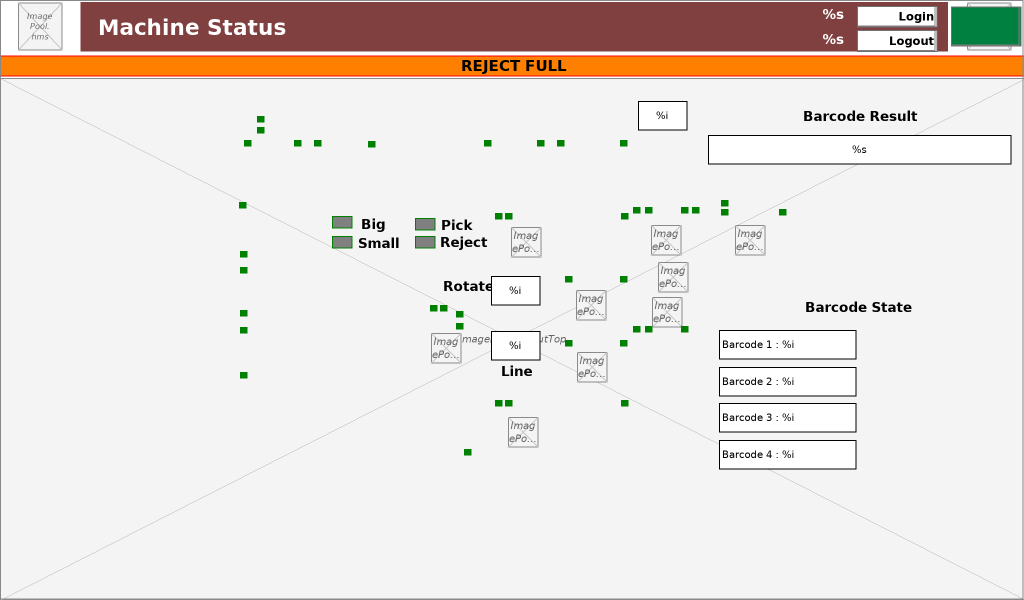
VISUALIZATION SeqStatus  // 1024x600
    Frame (0,-1 1024x55)
        shows Header()
    Label (95,15 250x25), "Machine Status"
    Image (0,78 1026x522), image: ImagePool.LayoutTop
    Image (431,333 30x30), image: ImagePool.info
        OnMouseDown: OpenDialog Dialog=PUSeq, OpenModal=True, OpenCentered=True
        OnMouseDown: execute { HMI_GVL.sCurrentJob :=  HMI_GVL.CJ_Picking; HMI_GVL.iSeqIndex   := HMI_GVL.SI_Picking; }
    Image (511,227 30x30), image: ImagePool.info
        OnMouseDown: OpenDialog Dialog=PUSeq, OpenModal=True, OpenCentered=True
        OnMouseDown: execute { HMI_GVL.sCurrentJob :=  HMI_GVL.CJ_Placing1; HMI_GVL.iSeqIndex   := HMI_GVL.SI_Placing1; }
    Image (576,290 30x30), image: ImagePool.info
        OnMouseDown: OpenDialog Dialog=PUSeq, OpenModal=True, OpenCentered=True
        OnMouseDown: execute { HMI_GVL.sCurrentJob :=  HMI_GVL.CJ_Placing2; HMI_GVL.iSeqIndex   := HMI_GVL.SI_Placing2; }
    Image (577,352 30x30), image: ImagePool.info
        OnMouseDown: OpenDialog Dialog=PUSeq, OpenModal=True, OpenCentered=True
        OnMouseDown: execute { HMI_GVL.sCurrentJob :=  HMI_GVL.CJ_Placing3; HMI_GVL.iSeqIndex   := HMI_GVL.SI_Placing3; }
    Image (508,417 30x30), image: ImagePool.info
        OnMouseDown: OpenDialog Dialog=PUSeq, OpenModal=True, OpenCentered=True
        OnMouseDown: execute { HMI_GVL.sCurrentJob :=  HMI_GVL.CJ_Placing4; HMI_GVL.iSeqIndex   := HMI_GVL.SI_Placing4; }
    Image (735,225 30x30), image: ImagePool.info
        OnMouseDown: OpenDialog Dialog=PUSeq, OpenModal=True, OpenCentered=True
        OnMouseDown: execute { HMI_GVL.sCurrentJob :=  HMI_GVL.CJ_Dispenser; HMI_GVL.iSeqIndex   := InputOutput_GVL.SeqIndexOutfeed[4]; }
    Image (652,297 30x30), image: ImagePool.info
        OnMouseDown: OpenDialog Dialog=PUSeq, OpenModal=True, OpenCentered=True
        OnMouseDown: execute { HMI_GVL.sCurrentJob :=  HMI_GVL.CJ_ShuttleEmpty; HMI_GVL.iSeqIndex   := InputOutput_GVL.SeqIndexOutfeed[1]; }
    Image (651,225 30x30), image: ImagePool.info
        OnMouseDown: OpenDialog Dialog=PUSeq, OpenModal=True, OpenCentered=True
        OnMouseDown: execute { HMI_GVL.sCurrentJob :=  HMI_GVL.CJ_ShuttleLoad; HMI_GVL.iSeqIndex   := InputOutput_GVL.SeqIndexOutfeed[2]; }
    Image (658,262 30x30), image: ImagePool.info
        OnMouseDown: OpenDialog Dialog=PUSeq, OpenModal=True, OpenCentered=True
        OnMouseDown: execute { HMI_GVL.sCurrentJob :=  HMI_GVL.CJ_ShuttleManagement; HMI_GVL.iSeqIndex   := InputOutput_GVL.SeqIndexOutfeed[3]; }
    Rectangle (415,218 20x12), colour toggle: InputOutput_GVL.xOut_Robot.Pick
    Rectangle (415,236 20x12), colour toggle: InputOutput_GVL.xOut_Robot.RejectBox
    Label (438,213 65x25), "Pick"
    Label (437,230 65x25), "Reject"
    Rectangle (456,323 7x6), colour toggle: InputOutput_GVL.xIn1405
    Rectangle (456,311 7x6), colour toggle: InputOutput_GVL.xIn1406
    Rectangle (430,305 7x6), colour toggle: InputOutput_GVL.xIn1407
    Rectangle (440,305 7x6), colour toggle: InputOutput_GVL.xIn1400
    Rectangle (633,207 7x6), colour toggle: InputOutput_GVL.Digital_Input[124]
    Rectangle (645,207 7x6), colour toggle: InputOutput_GVL.Digital_Input[122]
    Rectangle (681,207 7x6), colour toggle: InputOutput_GVL.Digital_Input[121]
    Rectangle (692,207 7x6), colour toggle: InputOutput_GVL.Digital_Input[123]
    Rectangle (633,326 7x6), colour toggle: InputOutput_GVL.Digital_Input[119]
    Rectangle (645,326 7x6), colour toggle: InputOutput_GVL.Digital_Input[117]
    Rectangle (681,326 7x6), colour toggle: InputOutput_GVL.Digital_Input[118]
    Rectangle (721,209 7x6), colour toggle: InputOutput_GVL.Digital_Input[51]
    Rectangle (721,200 7x6), colour toggle: InputOutput_GVL.Digital_Input[52]
    Rectangle (779,209 7x6), colour toggle: InputOutput_GVL.Digital_Input[50]
    Rectangle (495,400 7x6), colour toggle: InputOutput_GVL.xIn1509
    Rectangle (505,400 7x6), colour toggle: InputOutput_GVL.xIn1508
    Rectangle (621,400 7x6), colour toggle: InputOutput_GVL.xIn1507
    Rectangle (565,340 7x6), colour toggle: InputOutput_GVL.xIn1506
    Rectangle (620,340 7x6), colour toggle: InputOutput_GVL.xIn1505
    Rectangle (565,276 7x6), colour toggle: InputOutput_GVL.xIn1504
    Rectangle (620,276 7x6), colour toggle: InputOutput_GVL.xIn1503
    Rectangle (495,213 7x6), colour toggle: InputOutput_GVL.xIn1502
    Rectangle (505,213 7x6), colour toggle: InputOutput_GVL.xIn1501
    Rectangle (621,213 7x6), colour toggle: InputOutput_GVL.xIn1500
    Rectangle (620,140 7x6), colour toggle: InputOutput_GVL.Digital_Input[14]
    Rectangle (557,140 7x6), colour toggle: InputOutput_GVL.Digital_Input[15]
    Rectangle (537,140 7x6), colour toggle: InputOutput_GVL.Digital_Input[37]
    Rectangle (484,140 7x6), colour toggle: InputOutput_GVL.Digital_Input[38]
    Rectangle (368,141 7x6), colour toggle: InputOutput_GVL.Digital_Input[39]
    Rectangle (314,140 7x6), colour toggle: InputOutput_GVL.Digital_Input[40]
    Rectangle (294,140 7x6), colour toggle: InputOutput_GVL.Digital_Input[41]
    Rectangle (244,140 7x6), colour toggle: InputOutput_GVL.Digital_Input[42]
    Rectangle (239,202 7x6), colour toggle: InputOutput_GVL.Digital_Input[45]
    Rectangle (240,251 7x6), colour toggle: InputOutput_GVL.Digital_Input[46]
    Rectangle (240,267 7x6), colour toggle: InputOutput_GVL.Digital_Input[47]
    Rectangle (240,310 7x6), colour toggle: InputOutput_GVL.Digital_Input[48]
    Rectangle (240,327 7x6), colour toggle: InputOutput_GVL.Digital_Input[8]
    Rectangle (240,372 7x6), colour toggle: InputOutput_GVL.Digital_Input[9]
    Rectangle (257,127 7x6), colour toggle: InputOutput_GVL.Digital_Input[43]
    Rectangle (257,116 7x6), colour toggle: InputOutput_GVL.Digital_Input[44]
    Rectangle (464,449 7x6), colour toggle: InputOutput_GVL.xIn1005
    RoundedRectangle (638,101 49x29), "%i", text variable: InputOutput_GVL.ShuttlePosition
    Rectangle (332,216 20x12), colour toggle: InputOutput_GVL.xOut_Robot.CheckBigBox
    Label (358,212 65x25), "Big"
    Rectangle (332,236 20x12), colour toggle: InputOutput_GVL.xOut_Robot.CheckSmallBox
    Label (355,231 65x25), "Small"
    RoundedRectangle (708,135 303x29), "%s", text variable: Status_GVL.BarcodeResult
    Label (712,104 297x25), "Barcode Result"
    Label (710,295 297x25), "Barcode State"
    RoundedRectangle (719,330 137x29), "Barcode 1 : %i", text variable: InputOutput_GVL.BarcodeReader_Picking1_State
    RoundedRectangle (719,367 137x29), "Barcode 2 : %i", text variable: InputOutput_GVL.BarcodeReader_Picking2B_State
    RoundedRectangle (719,403 137x29), "Barcode 3 : %i", text variable: InputOutput_GVL.BarcodeReader_Picking3B_State
    RoundedRectangle (719,440 137x29), "Barcode 4 : %i", text variable: InputOutput_GVL.BarcodeReader_Picking4_State
    RoundedRectangle (491,331 49x29), "%i", text variable: HMI_GVL.PickLine
    Label (440,274 65x25), "Rotate"
    RoundedRectangle (491,276 49x29), "%i", text variable: InputOutput_GVL.xOut_Robot.RotatePickInt
    Label (498,359 65x25), "Line"
END_VISUALIZATION

// ---- VISUs/PLC Status/IO_Status.TcVIS
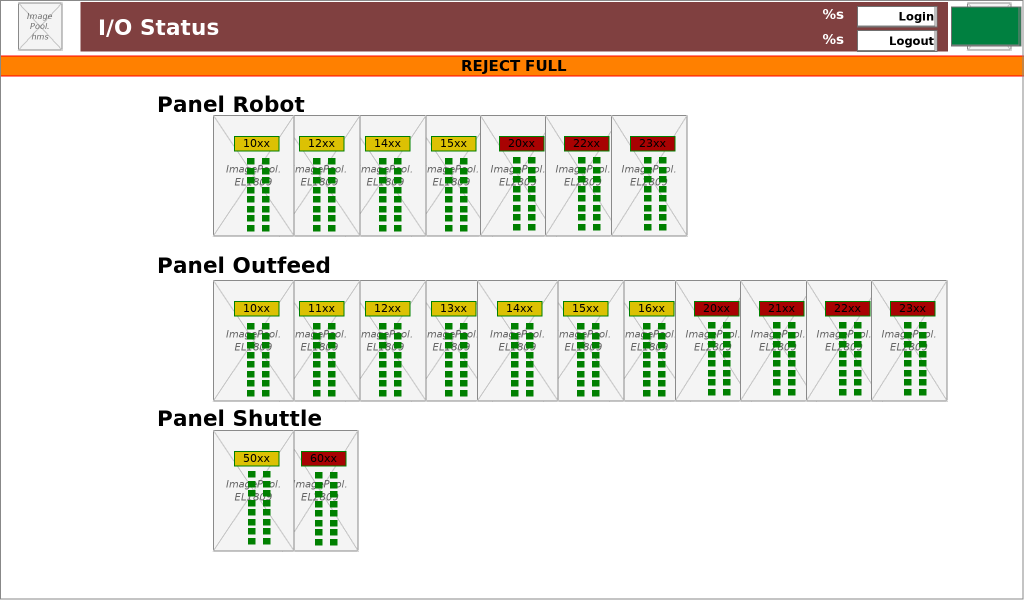
VISUALIZATION IO_Status  // 1024x600
    Image (282,430 76x121), image: ImagePool.EL2809
        OnMouseClick: OpenDialog Dialog=P3_DO1, OpenModal=True, OpenCentered=True
    Image (213,430 81x121), image: ImagePool.EL1809
        OnMouseClick: OpenDialog Dialog=P3_DI1, OpenModal=True, OpenCentered=True
    Image (411,115 81x121), image: ImagePool.EL1809
        OnMouseClick: OpenDialog Dialog=P1_DI4, OpenModal=True, OpenCentered=True
    Image (345,115 81x121), image: ImagePool.EL1809
        OnMouseClick: OpenDialog Dialog=P1_DI3, OpenModal=True, OpenCentered=True
    Image (279,115 81x121), image: ImagePool.EL1809
        OnMouseClick: OpenDialog Dialog=P1_DI2, OpenModal=True, OpenCentered=True
    Frame (0,-1 1024x55)
        shows Header()
    Label (95,15 250x25), "I/O Status"
    Image (213,115 81x121), image: ImagePool.EL1809
        OnMouseClick: OpenDialog Dialog=P1_DI1, OpenModal=True, OpenCentered=True
    Rectangle (247,158 7x6), colour toggle: InputOutput_GVL.xIn1000
    Rectangle (262,158 7x6), colour toggle: InputOutput_GVL.xIn1008
    Rectangle (247,168 7x6), colour toggle: InputOutput_GVL.xIn1001
    Rectangle (262,168 7x6), colour toggle: InputOutput_GVL.xIn1009
    Rectangle (247,177 7x6), colour toggle: InputOutput_GVL.xIn1002
    Rectangle (262,177 7x6), colour toggle: InputOutput_GVL.xIn1010
    Rectangle (247,187 7x6), colour toggle: InputOutput_GVL.xIn1003
    Rectangle (262,187 7x6), colour toggle: InputOutput_GVL.xIn1011
    Rectangle (247,196 7x6), colour toggle: InputOutput_GVL.xIn1004
    Rectangle (262,196 7x6), colour toggle: InputOutput_GVL.xIn1012
    Rectangle (247,206 7x6), colour toggle: InputOutput_GVL.xIn1005
    Rectangle (262,206 7x6), colour toggle: InputOutput_GVL.xIn1013
    Rectangle (247,215 7x6), colour toggle: InputOutput_GVL.xIn1006
    Rectangle (262,215 7x6), colour toggle: InputOutput_GVL.xIn1014
    Rectangle (247,225 7x6), colour toggle: InputOutput_GVL.xIn1007
    Rectangle (262,225 7x6), colour toggle: InputOutput_GVL.xIn1015
    Label (237,134 37x20), "10xx"
    Rectangle (313,158 7x6), colour toggle: InputOutput_GVL.xIn1200
    Rectangle (328,158 7x6), colour toggle: InputOutput_GVL.xIn1208
    Rectangle (313,168 7x6), colour toggle: InputOutput_GVL.xIn1201
    Rectangle (328,168 7x6), colour toggle: InputOutput_GVL.xIn1209
    Rectangle (313,177 7x6), colour toggle: InputOutput_GVL.xIn1202
    Rectangle (328,177 7x6), colour toggle: InputOutput_GVL.xIn1210
    Rectangle (313,187 7x6), colour toggle: InputOutput_GVL.xIn1203
    Rectangle (328,187 7x6), colour toggle: InputOutput_GVL.xIn1211
    Rectangle (313,196 7x6), colour toggle: InputOutput_GVL.xIn1204
    Rectangle (328,196 7x6), colour toggle: InputOutput_GVL.xIn1212
    Rectangle (313,206 7x6), colour toggle: InputOutput_GVL.xIn1205
    Rectangle (328,206 7x6), colour toggle: InputOutput_GVL.xIn1213
    Rectangle (313,215 7x6), colour toggle: InputOutput_GVL.xIn1206
    Rectangle (328,215 7x6), colour toggle: InputOutput_GVL.xIn1214
    Rectangle (313,225 7x6), colour toggle: InputOutput_GVL.xIn1207
    Rectangle (328,225 7x6), colour toggle: InputOutput_GVL.xIn1215
    Rectangle (379,158 7x6), colour toggle: InputOutput_GVL.xIn1400
    Rectangle (394,158 7x6), colour toggle: InputOutput_GVL.xIn1408
    Rectangle (379,168 7x6), colour toggle: InputOutput_GVL.xIn1401
    Rectangle (394,168 7x6), colour toggle: InputOutput_GVL.xIn1409
    Rectangle (379,177 7x6), colour toggle: InputOutput_GVL.xIn1402
    Rectangle (394,177 7x6), colour toggle: InputOutput_GVL.xIn1410
    Rectangle (379,187 7x6), colour toggle: InputOutput_GVL.xIn1403
    Rectangle (394,187 7x6), colour toggle: InputOutput_GVL.xIn1411
    Rectangle (379,196 7x6), colour toggle: InputOutput_GVL.xIn1404
    Rectangle (394,196 7x6), colour toggle: InputOutput_GVL.xIn1412
    Rectangle (379,206 7x6), colour toggle: InputOutput_GVL.xIn1405
    Rectangle (394,206 7x6), colour toggle: InputOutput_GVL.xIn1413
    Rectangle (379,215 7x6), colour toggle: InputOutput_GVL.xIn1406
    Rectangle (394,215 7x6), colour toggle: InputOutput_GVL.xIn1414
    Rectangle (379,225 7x6), colour toggle: InputOutput_GVL.xIn1407
    Rectangle (394,225 7x6), colour toggle: InputOutput_GVL.xIn1415
    Rectangle (445,158 7x6), colour toggle: InputOutput_GVL.xIn1500
    Rectangle (460,158 7x6), colour toggle: InputOutput_GVL.xIn1508
    Rectangle (445,168 7x6), colour toggle: InputOutput_GVL.xIn1501
    Rectangle (460,168 7x6), colour toggle: InputOutput_GVL.xIn1509
    Rectangle (445,177 7x6), colour toggle: InputOutput_GVL.xIn1502
    Rectangle (460,177 7x6), colour toggle: InputOutput_GVL.xIn1510
    Rectangle (445,187 7x6), colour toggle: InputOutput_GVL.xIn1503
    Rectangle (460,187 7x6), colour toggle: InputOutput_GVL.xIn1511
    Rectangle (445,196 7x6), colour toggle: InputOutput_GVL.xIn1504
    Rectangle (460,196 7x6), colour toggle: InputOutput_GVL.xIn1512
    Rectangle (445,206 7x6), colour toggle: InputOutput_GVL.xIn1505
    Rectangle (460,206 7x6), colour toggle: InputOutput_GVL.xIn1513
    Rectangle (445,215 7x6), colour toggle: InputOutput_GVL.xIn1506
    Rectangle (460,215 7x6), colour toggle: InputOutput_GVL.xIn1514
    Rectangle (445,225 7x6), colour toggle: InputOutput_GVL.xIn1507
    Rectangle (460,225 7x6), colour toggle: InputOutput_GVL.xIn1515
    Rectangle (234,136 45x15), "10xx", colour toggle: HMI_GVL.xOut_HMI_Status_EcSlave[1]
    Rectangle (299,136 45x15), "12xx", colour toggle: HMI_GVL.xOut_HMI_Status_EcSlave[2]
    Rectangle (365,136 45x15), "14xx", colour toggle: HMI_GVL.xOut_HMI_Status_EcSlave[3]
    Rectangle (431,136 45x15), "15xx", colour toggle: HMI_GVL.xOut_HMI_Status_EcSlave[4]
    Image (480,115 76x121), image: ImagePool.EL2809
        OnMouseClick: OpenDialog Dialog=P1_DO1, OpenModal=True, OpenCentered=True
    Rectangle (513,157 7x6), colour toggle: InputOutput_GVL.xOut2000
    Rectangle (528,157 7x6), colour toggle: InputOutput_GVL.xOut2008
    Rectangle (513,167 7x6), colour toggle: InputOutput_GVL.xOut2001
    Rectangle (528,167 7x6), colour toggle: InputOutput_GVL.xOut2009
    Rectangle (513,176 7x6), colour toggle: InputOutput_GVL.xOut2002
    Rectangle (528,176 7x6), colour toggle: InputOutput_GVL.xOut2010
    Rectangle (513,186 7x6), colour toggle: InputOutput_GVL.xOut2003
    Rectangle (528,186 7x6), colour toggle: InputOutput_GVL.xOut2011
    Rectangle (513,195 7x6), colour toggle: InputOutput_GVL.xOut2004
    Rectangle (528,195 7x6), colour toggle: InputOutput_GVL.xOut2012
    Rectangle (513,205 7x6), colour toggle: InputOutput_GVL.xOut2005
    Rectangle (528,205 7x6), colour toggle: InputOutput_GVL.xOut2013
    Rectangle (513,214 7x6), colour toggle: InputOutput_GVL.xOut2006
    Rectangle (528,214 7x6), colour toggle: InputOutput_GVL.xOut2014
    Rectangle (513,224 7x6), colour toggle: InputOutput_GVL.xOut2007
    Rectangle (528,224 7x6), colour toggle: InputOutput_GVL.xOut2015
    Label (502,136 37x20), "10xx"
    Rectangle (499,136 45x15), "20xx", colour toggle: HMI_GVL.xOut_HMI_Status_EcSlave[5]
    Image (545,115 76x121), image: ImagePool.EL2809
        OnMouseClick: OpenDialog Dialog=P1_DO2, OpenModal=True, OpenCentered=True
    Rectangle (578,157 7x6), colour toggle: InputOutput_GVL.xOut2200
    Rectangle (593,157 7x6), colour toggle: InputOutput_GVL.xOut2208
    Rectangle (578,167 7x6), colour toggle: InputOutput_GVL.xOut2201
    Rectangle (593,167 7x6), colour toggle: InputOutput_GVL.xOut2209
    Rectangle (578,176 7x6), colour toggle: InputOutput_GVL.xOut2202
    Rectangle (593,176 7x6), colour toggle: InputOutput_GVL.xOut2210
    Rectangle (578,186 7x6), colour toggle: InputOutput_GVL.xOut2203
    Rectangle (593,186 7x6), colour toggle: InputOutput_GVL.xOut2211
    Rectangle (578,195 7x6), colour toggle: InputOutput_GVL.xOut2204
    Rectangle (593,195 7x6), colour toggle: InputOutput_GVL.xOut2212
    Rectangle (578,205 7x6), colour toggle: InputOutput_GVL.xOut2205
    Rectangle (593,205 7x6), colour toggle: InputOutput_GVL.xOut2213
    Rectangle (578,214 7x6), colour toggle: InputOutput_GVL.xOut2206
    Rectangle (593,214 7x6), colour toggle: InputOutput_GVL.xOut2214
    Rectangle (578,224 7x6), colour toggle: InputOutput_GVL.xOut2207
    Rectangle (593,224 7x6), colour toggle: InputOutput_GVL.xOut2215
    Label (567,135 37x20), "10xx"
    Rectangle (564,136 45x15), "22xx", colour toggle: HMI_GVL.xOut_HMI_Status_EcSlave[6]
    Image (611,115 76x121), image: ImagePool.EL2809
        OnMouseClick: OpenDialog Dialog=P1_DO3, OpenModal=True, OpenCentered=True
    Rectangle (644,157 7x6), colour toggle: InputOutput_GVL.xOut2300
    Rectangle (659,157 7x6), colour toggle: InputOutput_GVL.xOut2308
    Rectangle (644,167 7x6), colour toggle: InputOutput_GVL.xOut2301
    Rectangle (659,167 7x6), colour toggle: InputOutput_GVL.xOut2309
    Rectangle (644,176 7x6), colour toggle: InputOutput_GVL.xOut2302
    Rectangle (659,176 7x6), colour toggle: InputOutput_GVL.xOut2310
    Rectangle (644,186 7x6), colour toggle: InputOutput_GVL.xOut2303
    Rectangle (659,186 7x6), colour toggle: InputOutput_GVL.xOut2311
    Rectangle (644,195 7x6), colour toggle: InputOutput_GVL.xOut2304
    Rectangle (659,195 7x6), colour toggle: InputOutput_GVL.xOut2312
    Rectangle (644,205 7x6), colour toggle: InputOutput_GVL.xOut2305
    Rectangle (659,205 7x6), colour toggle: InputOutput_GVL.xOut2313
    Rectangle (644,214 7x6), colour toggle: InputOutput_GVL.xOut2306
    Rectangle (659,214 7x6), colour toggle: InputOutput_GVL.xOut2314
    Rectangle (644,224 7x6), colour toggle: InputOutput_GVL.xOut2307
    Rectangle (659,224 7x6), colour toggle: InputOutput_GVL.xOut2315
    Label (633,135 37x20), "10xx"
    Rectangle (630,136 45x15), "23xx", colour toggle: HMI_GVL.xOut_HMI_Status_EcSlave[7]
    Label (154,92 250x25), "Panel Robot"
    Label (154,253 250x25), "Panel Outfeed"
    Rectangle (248,471 7x6), colour toggle: InputOutput_GVL.Digital_Input[113]
    Rectangle (263,471 7x6), colour toggle: InputOutput_GVL.Digital_Input[121]
    Rectangle (248,481 7x6), colour toggle: InputOutput_GVL.Digital_Input[114]
    Rectangle (263,481 7x6), colour toggle: InputOutput_GVL.Digital_Input[122]
    Rectangle (248,490 7x6), colour toggle: InputOutput_GVL.Digital_Input[115]
    Rectangle (263,490 7x6), colour toggle: InputOutput_GVL.Digital_Input[123]
    Rectangle (248,500 7x6), colour toggle: InputOutput_GVL.Digital_Input[116]
    Rectangle (263,500 7x6), colour toggle: InputOutput_GVL.Digital_Input[124]
    Rectangle (248,509 7x6), colour toggle: InputOutput_GVL.Digital_Input[117]
    Rectangle (263,509 7x6), colour toggle: InputOutput_GVL.Digital_Input[125]
    Rectangle (248,519 7x6), colour toggle: InputOutput_GVL.Digital_Input[118]
    Rectangle (263,519 7x6), colour toggle: InputOutput_GVL.Digital_Input[126]
    Rectangle (248,528 7x6), colour toggle: InputOutput_GVL.Digital_Input[119]
    Rectangle (263,528 7x6), colour toggle: InputOutput_GVL.Digital_Input[127]
    Rectangle (248,538 7x6), colour toggle: InputOutput_GVL.Digital_Input[120]
    Rectangle (263,538 7x6), colour toggle: InputOutput_GVL.Digital_Input[128]
    Label (237,448 37x20), "10xx"
    Rectangle (234,451 45x15), "50xx", colour toggle: HMI_GVL.xOut_HMI_Status_EcSlave[1]
    Rectangle (315,472 7x6), colour toggle: InputOutput_GVL.Digital_Output[65]
    Rectangle (330,472 7x6), colour toggle: InputOutput_GVL.Digital_Output[73]
    Rectangle (315,482 7x6), colour toggle: InputOutput_GVL.Digital_Output[66]
    Rectangle (330,482 7x6), colour toggle: InputOutput_GVL.Digital_Output[74]
    Rectangle (315,491 7x6), colour toggle: InputOutput_GVL.Digital_Output[67]
    Rectangle (330,491 7x6), colour toggle: InputOutput_GVL.Digital_Output[75]
    Rectangle (315,501 7x6), colour toggle: InputOutput_GVL.Digital_Output[68]
    Rectangle (330,501 7x6), colour toggle: InputOutput_GVL.Digital_Output[76]
    Rectangle (315,510 7x6), colour toggle: InputOutput_GVL.Digital_Output[69]
    Rectangle (330,510 7x6), colour toggle: InputOutput_GVL.Digital_Output[77]
    Rectangle (315,520 7x6), colour toggle: InputOutput_GVL.Digital_Output[70]
    Rectangle (330,520 7x6), colour toggle: InputOutput_GVL.Digital_Output[78]
    Rectangle (315,529 7x6), colour toggle: InputOutput_GVL.Digital_Output[71]
    Rectangle (330,529 7x6), colour toggle: InputOutput_GVL.Digital_Output[79]
    Rectangle (315,539 7x6), colour toggle: InputOutput_GVL.Digital_Output[72]
    Rectangle (330,539 7x6), colour toggle: InputOutput_GVL.Digital_Output[80]
    Label (304,450 37x20), "10xx"
    Rectangle (301,451 45x15), "60xx", colour toggle: HMI_GVL.xOut_HMI_Status_EcSlave[1]
    Label (154,406 250x25), "Panel Shuttle"
    Image (411,280 81x121), image: ImagePool.EL1809
        OnMouseClick: OpenDialog Dialog=P2_DI4, OpenModal=True, OpenCentered=True
    Image (345,280 81x121), image: ImagePool.EL1809
        OnMouseClick: OpenDialog Dialog=P2_DI3, OpenModal=True, OpenCentered=True
    Image (279,280 81x121), image: ImagePool.EL1809
        OnMouseClick: OpenDialog Dialog=P2_DI2, OpenModal=True, OpenCentered=True
    Image (213,280 81x121), image: ImagePool.EL1809
        OnMouseClick: OpenDialog Dialog=P2_DI1, OpenModal=True, OpenCentered=True
    Rectangle (247,323 7x6), colour toggle: InputOutput_GVL.Digital_Input[1]
    Rectangle (262,323 7x6), colour toggle: InputOutput_GVL.Digital_Input[9]
    Rectangle (247,333 7x6), colour toggle: InputOutput_GVL.Digital_Input[2]
    Rectangle (262,333 7x6), colour toggle: InputOutput_GVL.Digital_Input[10]
    Rectangle (247,342 7x6), colour toggle: InputOutput_GVL.Digital_Input[3]
    Rectangle (262,342 7x6), colour toggle: InputOutput_GVL.Digital_Input[11]
    Rectangle (247,352 7x6), colour toggle: InputOutput_GVL.Digital_Input[4]
    Rectangle (262,352 7x6), colour toggle: InputOutput_GVL.Digital_Input[12]
    Rectangle (247,361 7x6), colour toggle: InputOutput_GVL.Digital_Input[5]
    Rectangle (262,361 7x6), colour toggle: InputOutput_GVL.Digital_Input[13]
    Rectangle (247,371 7x6), colour toggle: InputOutput_GVL.Digital_Input[6]
    Rectangle (262,371 7x6), colour toggle: InputOutput_GVL.Digital_Input[14]
    Rectangle (247,380 7x6), colour toggle: InputOutput_GVL.Digital_Input[7]
    Rectangle (262,380 7x6), colour toggle: InputOutput_GVL.Digital_Input[15]
    Rectangle (247,390 7x6), colour toggle: InputOutput_GVL.Digital_Input[8]
    Rectangle (262,390 7x6), colour toggle: InputOutput_GVL.Digital_Input[16]
    Label (237,299 37x20), "10xx"
    Rectangle (313,323 7x6), colour toggle: InputOutput_GVL.Digital_Input[17]
    Rectangle (328,323 7x6), colour toggle: InputOutput_GVL.Digital_Input[25]
    Rectangle (313,333 7x6), colour toggle: InputOutput_GVL.Digital_Input[18]
    Rectangle (328,333 7x6), colour toggle: InputOutput_GVL.Digital_Input[26]
    Rectangle (313,342 7x6), colour toggle: InputOutput_GVL.Digital_Input[19]
    Rectangle (328,342 7x6), colour toggle: InputOutput_GVL.Digital_Input[27]
    Rectangle (313,352 7x6), colour toggle: InputOutput_GVL.Digital_Input[20]
    Rectangle (328,352 7x6), colour toggle: InputOutput_GVL.Digital_Input[28]
    Rectangle (313,361 7x6), colour toggle: InputOutput_GVL.Digital_Input[21]
    Rectangle (328,361 7x6), colour toggle: InputOutput_GVL.Digital_Input[29]
    Rectangle (313,371 7x6), colour toggle: InputOutput_GVL.Digital_Input[22]
    Rectangle (328,371 7x6), colour toggle: InputOutput_GVL.Digital_Input[30]
    Rectangle (313,380 7x6), colour toggle: InputOutput_GVL.Digital_Input[23]
    Rectangle (328,380 7x6), colour toggle: InputOutput_GVL.Digital_Input[31]
    Rectangle (313,390 7x6), colour toggle: InputOutput_GVL.Digital_Input[24]
    Rectangle (328,390 7x6), colour toggle: InputOutput_GVL.Digital_Input[32]
    Rectangle (379,323 7x6), colour toggle: InputOutput_GVL.Digital_Input[33]
    Rectangle (394,323 7x6), colour toggle: InputOutput_GVL.Digital_Input[41]
    Rectangle (379,333 7x6), colour toggle: InputOutput_GVL.Digital_Input[34]
    Rectangle (394,333 7x6), colour toggle: InputOutput_GVL.Digital_Input[42]
    Rectangle (379,342 7x6), colour toggle: InputOutput_GVL.Digital_Input[35]
    Rectangle (394,342 7x6), colour toggle: InputOutput_GVL.Digital_Input[43]
    Rectangle (379,352 7x6), colour toggle: InputOutput_GVL.Digital_Input[36]
    Rectangle (394,352 7x6), colour toggle: InputOutput_GVL.Digital_Input[44]
    Rectangle (379,361 7x6), colour toggle: InputOutput_GVL.Digital_Input[37]
    Rectangle (394,361 7x6), colour toggle: InputOutput_GVL.Digital_Input[45]
    Rectangle (379,371 7x6), colour toggle: InputOutput_GVL.Digital_Input[38]
    Rectangle (394,371 7x6), colour toggle: InputOutput_GVL.Digital_Input[46]
    Rectangle (379,380 7x6), colour toggle: InputOutput_GVL.Digital_Input[39]
    Rectangle (394,380 7x6), colour toggle: InputOutput_GVL.Digital_Input[47]
    Rectangle (379,390 7x6), colour toggle: InputOutput_GVL.Digital_Input[40]
    Rectangle (394,390 7x6), colour toggle: InputOutput_GVL.Digital_Input[48]
    Rectangle (445,323 7x6), colour toggle: InputOutput_GVL.Digital_Input[49]
    Rectangle (460,323 7x6), colour toggle: InputOutput_GVL.Digital_Input[57]
    Rectangle (445,333 7x6), colour toggle: InputOutput_GVL.Digital_Input[50]
    Rectangle (460,333 7x6), colour toggle: InputOutput_GVL.Digital_Input[58]
    Rectangle (445,342 7x6), colour toggle: InputOutput_GVL.Digital_Input[51]
    Rectangle (460,342 7x6), colour toggle: InputOutput_GVL.Digital_Input[59]
    Rectangle (445,352 7x6), colour toggle: InputOutput_GVL.Digital_Input[52]
    Rectangle (460,352 7x6), colour toggle: InputOutput_GVL.Digital_Input[60]
    Rectangle (445,361 7x6), colour toggle: InputOutput_GVL.Digital_Input[53]
    Rectangle (460,361 7x6), colour toggle: InputOutput_GVL.Digital_Input[61]
    Rectangle (445,371 7x6), colour toggle: InputOutput_GVL.Digital_Input[54]
    Rectangle (460,371 7x6), colour toggle: InputOutput_GVL.Digital_Input[62]
    Rectangle (445,380 7x6), colour toggle: InputOutput_GVL.Digital_Input[55]
    Rectangle (460,380 7x6), colour toggle: InputOutput_GVL.Digital_Input[63]
    Rectangle (445,390 7x6), colour toggle: InputOutput_GVL.Digital_Input[56]
    Rectangle (460,390 7x6), colour toggle: InputOutput_GVL.Digital_Input[64]
    Rectangle (234,301 45x15), "10xx", colour toggle: HMI_GVL.xOut_HMI_Status_EcSlave[1]
    Rectangle (299,301 45x15), "11xx", colour toggle: HMI_GVL.xOut_HMI_Status_EcSlave[2]
    Rectangle (365,301 45x15), "12xx", colour toggle: HMI_GVL.xOut_HMI_Status_EcSlave[3]
    Rectangle (431,301 45x15), "13xx", colour toggle: HMI_GVL.xOut_HMI_Status_EcSlave[4]
    Image (609,280 81x121), image: ImagePool.EL1809
        OnMouseClick: OpenDialog Dialog=P2_DI7, OpenModal=True, OpenCentered=True
    Image (543,280 81x121), image: ImagePool.EL1809
        OnMouseClick: OpenDialog Dialog=P2_DI6, OpenModal=True, OpenCentered=True
    Image (477,280 81x121), image: ImagePool.EL1809
        OnMouseClick: OpenDialog Dialog=P2_DI5, OpenModal=True, OpenCentered=True
    Rectangle (511,323 7x6), colour toggle: InputOutput_GVL.Digital_Input[65]
    Rectangle (526,323 7x6), colour toggle: InputOutput_GVL.Digital_Input[73]
    Rectangle (511,333 7x6), colour toggle: InputOutput_GVL.Digital_Input[66]
    Rectangle (526,333 7x6), colour toggle: InputOutput_GVL.Digital_Input[74]
    Rectangle (511,342 7x6), colour toggle: InputOutput_GVL.Digital_Input[67]
    Rectangle (526,342 7x6), colour toggle: InputOutput_GVL.Digital_Input[75]
    Rectangle (511,352 7x6), colour toggle: InputOutput_GVL.Digital_Input[68]
    Rectangle (526,352 7x6), colour toggle: InputOutput_GVL.Digital_Input[76]
    Rectangle (511,361 7x6), colour toggle: InputOutput_GVL.Digital_Input[69]
    Rectangle (526,361 7x6), colour toggle: InputOutput_GVL.Digital_Input[77]
    Rectangle (511,371 7x6), colour toggle: InputOutput_GVL.Digital_Input[70]
    Rectangle (526,371 7x6), colour toggle: InputOutput_GVL.Digital_Input[78]
    Rectangle (511,380 7x6), colour toggle: InputOutput_GVL.Digital_Input[71]
    Rectangle (526,380 7x6), colour toggle: InputOutput_GVL.Digital_Input[79]
    Rectangle (511,390 7x6), colour toggle: InputOutput_GVL.Digital_Input[72]
    Rectangle (526,390 7x6), colour toggle: InputOutput_GVL.Digital_Input[80]
    Rectangle (577,323 7x6), colour toggle: InputOutput_GVL.Digital_Input[81]
    Rectangle (592,323 7x6), colour toggle: InputOutput_GVL.Digital_Input[89]
    Rectangle (577,333 7x6), colour toggle: InputOutput_GVL.Digital_Input[82]
    Rectangle (592,333 7x6), colour toggle: InputOutput_GVL.Digital_Input[90]
    Rectangle (577,342 7x6), colour toggle: InputOutput_GVL.Digital_Input[83]
    Rectangle (592,342 7x6), colour toggle: InputOutput_GVL.Digital_Input[91]
    Rectangle (577,352 7x6), colour toggle: InputOutput_GVL.Digital_Input[84]
    Rectangle (592,352 7x6), colour toggle: InputOutput_GVL.Digital_Input[92]
    Rectangle (577,361 7x6), colour toggle: InputOutput_GVL.Digital_Input[85]
    Rectangle (592,361 7x6), colour toggle: InputOutput_GVL.Digital_Input[93]
    Rectangle (577,371 7x6), colour toggle: InputOutput_GVL.Digital_Input[86]
    Rectangle (592,371 7x6), colour toggle: InputOutput_GVL.Digital_Input[94]
    Rectangle (577,380 7x6), colour toggle: InputOutput_GVL.Digital_Input[87]
    Rectangle (592,380 7x6), colour toggle: InputOutput_GVL.Digital_Input[95]
    Rectangle (577,390 7x6), colour toggle: InputOutput_GVL.Digital_Input[88]
    Rectangle (592,390 7x6), colour toggle: InputOutput_GVL.Digital_Input[96]
    Rectangle (643,323 7x6), colour toggle: InputOutput_GVL.Digital_Input[97]
    Rectangle (658,323 7x6), colour toggle: InputOutput_GVL.Digital_Input[105]
    Rectangle (643,333 7x6), colour toggle: InputOutput_GVL.Digital_Input[98]
    Rectangle (658,333 7x6), colour toggle: InputOutput_GVL.Digital_Input[106]
    Rectangle (643,342 7x6), colour toggle: InputOutput_GVL.Digital_Input[99]
    Rectangle (658,342 7x6), colour toggle: InputOutput_GVL.Digital_Input[107]
    Rectangle (643,352 7x6), colour toggle: InputOutput_GVL.Digital_Input[100]
    Rectangle (658,352 7x6), colour toggle: InputOutput_GVL.Digital_Input[108]
    Rectangle (643,361 7x6), colour toggle: InputOutput_GVL.Digital_Input[101]
    Rectangle (658,361 7x6), colour toggle: InputOutput_GVL.Digital_Input[109]
    Rectangle (643,371 7x6), colour toggle: InputOutput_GVL.Digital_Input[102]
    Rectangle (658,371 7x6), colour toggle: InputOutput_GVL.Digital_Input[110]
    Rectangle (643,380 7x6), colour toggle: InputOutput_GVL.Digital_Input[103]
    Rectangle (658,380 7x6), colour toggle: InputOutput_GVL.Digital_Input[111]
    Rectangle (643,390 7x6), colour toggle: InputOutput_GVL.Digital_Input[104]
    Rectangle (658,390 7x6), colour toggle: InputOutput_GVL.Digital_Input[112]
    Rectangle (497,301 45x15), "14xx", colour toggle: HMI_GVL.xOut_HMI_Status_EcSlave[2]
    Rectangle (563,301 45x15), "15xx", colour toggle: HMI_GVL.xOut_HMI_Status_EcSlave[3]
    Rectangle (629,301 45x15), "16xx", colour toggle: HMI_GVL.xOut_HMI_Status_EcSlave[4]
    Image (675,280 76x121), image: ImagePool.EL2809
        OnMouseClick: OpenDialog Dialog=P2_DO1, OpenModal=True, OpenCentered=True
    Rectangle (708,322 7x6), colour toggle: InputOutput_GVL.Digital_Output[1]
    Rectangle (723,322 7x6), colour toggle: InputOutput_GVL.Digital_Output[9]
    Rectangle (708,332 7x6), colour toggle: InputOutput_GVL.Digital_Output[2]
    Rectangle (723,332 7x6), colour toggle: InputOutput_GVL.Digital_Output[10]
    Rectangle (708,341 7x6), colour toggle: InputOutput_GVL.Digital_Output[3]
    Rectangle (723,341 7x6), colour toggle: InputOutput_GVL.Digital_Output[11]
    Rectangle (708,351 7x6), colour toggle: InputOutput_GVL.Digital_Output[4]
    Rectangle (723,351 7x6), colour toggle: InputOutput_GVL.Digital_Output[12]
    Rectangle (708,360 7x6), colour toggle: InputOutput_GVL.Digital_Output[5]
    Rectangle (723,360 7x6), colour toggle: InputOutput_GVL.Digital_Output[13]
    Rectangle (708,370 7x6), colour toggle: InputOutput_GVL.Digital_Output[6]
    Rectangle (723,370 7x6), colour toggle: InputOutput_GVL.Digital_Output[14]
    Rectangle (708,379 7x6), colour toggle: InputOutput_GVL.Digital_Output[7]
    Rectangle (723,379 7x6), colour toggle: InputOutput_GVL.Digital_Output[15]
    Rectangle (708,389 7x6), colour toggle: InputOutput_GVL.Digital_Output[8]
    Rectangle (723,389 7x6), colour toggle: InputOutput_GVL.Digital_Output[16]
    Label (697,301 37x20), "10xx"
    Rectangle (694,301 45x15), "20xx", colour toggle: HMI_GVL.xOut_HMI_Status_EcSlave[1]
    Image (740,280 76x121), image: ImagePool.EL2809
        OnMouseClick: OpenDialog Dialog=P2_DO2, OpenModal=True, OpenCentered=True
    Rectangle (773,322 7x6), colour toggle: InputOutput_GVL.Digital_Output[17]
    Rectangle (788,322 7x6), colour toggle: InputOutput_GVL.Digital_Output[25]
    Rectangle (773,332 7x6), colour toggle: InputOutput_GVL.Digital_Output[18]
    Rectangle (788,332 7x6), colour toggle: InputOutput_GVL.Digital_Output[26]
    Rectangle (773,341 7x6), colour toggle: InputOutput_GVL.Digital_Output[19]
    Rectangle (788,341 7x6), colour toggle: InputOutput_GVL.Digital_Output[27]
    Rectangle (773,351 7x6), colour toggle: InputOutput_GVL.Digital_Output[20]
    Rectangle (788,351 7x6), colour toggle: InputOutput_GVL.Digital_Output[28]
    Rectangle (773,360 7x6), colour toggle: InputOutput_GVL.Digital_Output[21]
    Rectangle (788,360 7x6), colour toggle: InputOutput_GVL.Digital_Output[29]
    Rectangle (773,370 7x6), colour toggle: InputOutput_GVL.Digital_Output[22]
    Rectangle (788,370 7x6), colour toggle: InputOutput_GVL.Digital_Output[30]
    Rectangle (773,379 7x6), colour toggle: InputOutput_GVL.Digital_Output[23]
    Rectangle (788,379 7x6), colour toggle: InputOutput_GVL.Digital_Output[31]
    Rectangle (773,389 7x6), colour toggle: InputOutput_GVL.Digital_Output[24]
    Rectangle (788,389 7x6), colour toggle: InputOutput_GVL.Digital_Output[32]
    Label (762,300 37x20), "10xx"
    Rectangle (759,301 45x15), "21xx", colour toggle: HMI_GVL.xOut_HMI_Status_EcSlave[1]
    Image (806,280 76x121), image: ImagePool.EL2809
        OnMouseClick: OpenDialog Dialog=P2_DO3, OpenModal=True, OpenCentered=True
    Rectangle (839,322 7x6), colour toggle: InputOutput_GVL.Digital_Output[33]
    Rectangle (854,322 7x6), colour toggle: InputOutput_GVL.Digital_Output[41]
    Rectangle (839,332 7x6), colour toggle: InputOutput_GVL.Digital_Output[34]
    Rectangle (854,332 7x6), colour toggle: InputOutput_GVL.Digital_Output[42]
    Rectangle (839,341 7x6), colour toggle: InputOutput_GVL.Digital_Output[35]
    Rectangle (854,341 7x6), colour toggle: InputOutput_GVL.Digital_Output[43]
    Rectangle (839,351 7x6), colour toggle: InputOutput_GVL.Digital_Output[36]
    Rectangle (854,351 7x6), colour toggle: InputOutput_GVL.Digital_Output[44]
    Rectangle (839,360 7x6), colour toggle: InputOutput_GVL.Digital_Output[37]
    Rectangle (854,360 7x6), colour toggle: InputOutput_GVL.Digital_Output[45]
    Rectangle (839,370 7x6), colour toggle: InputOutput_GVL.Digital_Output[38]
    Rectangle (854,370 7x6), colour toggle: InputOutput_GVL.Digital_Output[46]
    Rectangle (839,379 7x6), colour toggle: InputOutput_GVL.Digital_Output[39]
    Rectangle (854,379 7x6), colour toggle: InputOutput_GVL.Digital_Output[47]
    Rectangle (839,389 7x6), colour toggle: InputOutput_GVL.Digital_Output[40]
    Rectangle (854,389 7x6), colour toggle: InputOutput_GVL.Digital_Output[48]
    Label (828,300 37x20), "10xx"
    Rectangle (825,301 45x15), "22xx", colour toggle: HMI_GVL.xOut_HMI_Status_EcSlave[1]
    Image (871,280 76x121), image: ImagePool.EL2809
        OnMouseClick: OpenDialog Dialog=P2_DO4, OpenModal=True, OpenCentered=True
    Rectangle (904,322 7x6), colour toggle: InputOutput_GVL.Digital_Output[49]
    Rectangle (919,322 7x6), colour toggle: InputOutput_GVL.Digital_Output[57]
    Rectangle (904,332 7x6), colour toggle: InputOutput_GVL.Digital_Output[50]
    Rectangle (919,332 7x6), colour toggle: InputOutput_GVL.Digital_Output[58]
    Rectangle (904,341 7x6), colour toggle: InputOutput_GVL.Digital_Output[51]
    Rectangle (919,341 7x6), colour toggle: InputOutput_GVL.Digital_Output[59]
    Rectangle (904,351 7x6), colour toggle: InputOutput_GVL.Digital_Output[52]
    Rectangle (919,351 7x6), colour toggle: InputOutput_GVL.Digital_Output[60]
    Rectangle (904,360 7x6), colour toggle: InputOutput_GVL.Digital_Output[53]
    Rectangle (919,360 7x6), colour toggle: InputOutput_GVL.Digital_Output[61]
    Rectangle (904,370 7x6), colour toggle: InputOutput_GVL.Digital_Output[54]
    Rectangle (919,370 7x6), colour toggle: InputOutput_GVL.Digital_Output[62]
    Rectangle (904,379 7x6), colour toggle: InputOutput_GVL.Digital_Output[55]
    Rectangle (919,379 7x6), colour toggle: InputOutput_GVL.Digital_Output[63]
    Rectangle (904,389 7x6), colour toggle: InputOutput_GVL.Digital_Output[56]
    Rectangle (919,389 7x6), colour toggle: InputOutput_GVL.Digital_Output[64]
    Label (893,300 37x20), "10xx"
    Rectangle (890,301 45x15), "23xx", colour toggle: HMI_GVL.xOut_HMI_Status_EcSlave[1]
END_VISUALIZATION

// ---- VISUs/TestMode/Test_Outfeed.TcVIS
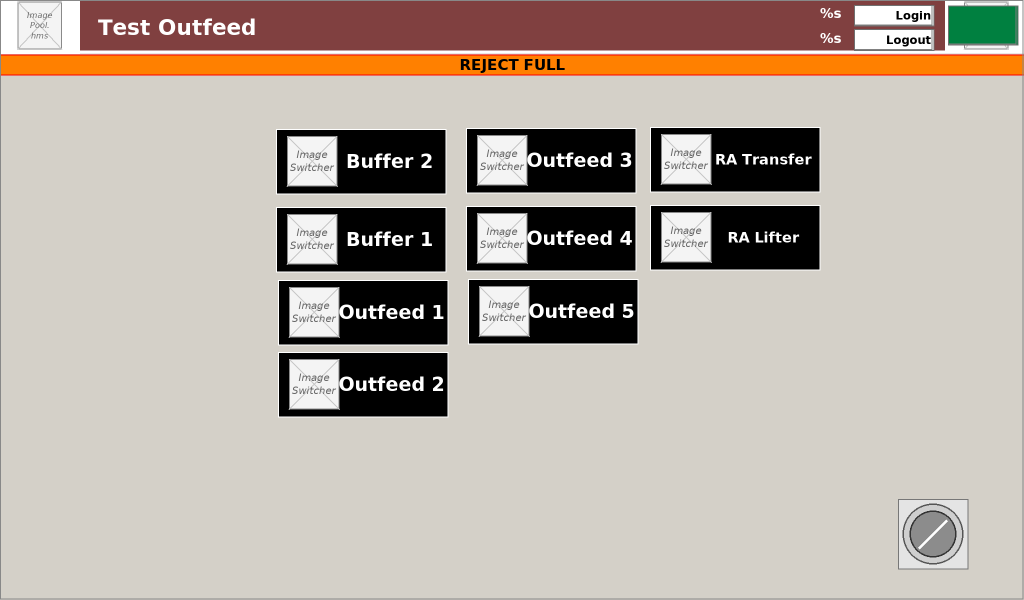
VISUALIZATION Test_Outfeed  // 1024x600
    Frame (0,-2 1021x55)
        shows Header()
    Label (95,15 250x25), "Test Outfeed"
    RotarySwitch (898,499 70x70), variable: HMI_GVL.bTestModeEnableOutfeed, behaviour: TOGGLE, style: Switch-RotarySwitch-Gray
    Group (276,129 182x65)
        toggle HMI_GVL.Test_PalletBuffer2_Fwd
        RoundedRectangle (0,0 170x65)
        Label (45,20 137x25), "Buffer 2"
        ImageSwitcher (11,7 50x50), variable: HMI_GVL.Test_PalletBuffer2_Fwd, behaviour: TOGGLE
    RoundedRectangle (276,207 170x65)
        toggle HMI_GVL.Test_PalletBuffer1_Fwd
    Label (321,227 137x25), "Buffer 1"
    ImageSwitcher (287,214 50x50), variable: HMI_GVL.Test_PalletBuffer1_Fwd, behaviour: TOGGLE
    RoundedRectangle (278,280 170x65)
        toggle HMI_GVL.Test_PalletOutfeed1_Fwd
    Label (323,300 137x25), "Outfeed 1"
    ImageSwitcher (289,287 50x50), variable: HMI_GVL.Test_PalletOutfeed1_Fwd, behaviour: TOGGLE
    RoundedRectangle (278,352 170x65)
        toggle HMI_GVL.Test_PalletOutfeed2_Fwd
    Label (323,372 137x25), "Outfeed 2"
    ImageSwitcher (289,359 50x50), variable: HMI_GVL.Test_PalletOutfeed2_Fwd, behaviour: TOGGLE
    RoundedRectangle (466,128 170x65)
        toggle HMI_GVL.Test_PalletOutfeed3_Fwd
    Label (511,148 137x25), "Outfeed 3"
    ImageSwitcher (477,135 50x50), variable: HMI_GVL.Test_PalletOutfeed3_Fwd, behaviour: TOGGLE
    RoundedRectangle (466,206 170x65)
        toggle HMI_GVL.Test_PalletOutfeed4_Fwd
    Label (511,226 137x25), "Outfeed 4"
    ImageSwitcher (477,213 50x50), variable: HMI_GVL.Test_PalletOutfeed4_Fwd, behaviour: TOGGLE
    RoundedRectangle (468,279 170x65)
        toggle HMI_GVL.Test_PalletOutfeed5_Fwd
    Label (513,299 137x25), "Outfeed 5"
    ImageSwitcher (479,286 50x50), variable: HMI_GVL.Test_PalletOutfeed5_Fwd, behaviour: TOGGLE
    RoundedRectangle (650,127 170x65)
        toggle HMI_GVL.Test_PalletRATransfer
    Label (695,147 137x25), "RA Transfer"
    ImageSwitcher (661,134 50x50), variable: HMI_GVL.Test_PalletRATransfer, behaviour: TOGGLE
    RoundedRectangle (650,205 170x65)
        tap HMI_GVL.Test_PalletRALifter
    Label (695,225 137x25), "RA Lifter"
    ImageSwitcher (661,212 50x50), variable: HMI_GVL.Test_PalletRALifter, behaviour: TOGGLE
END_VISUALIZATION

// ---- VISUs/TestMode/Control.TcVIS
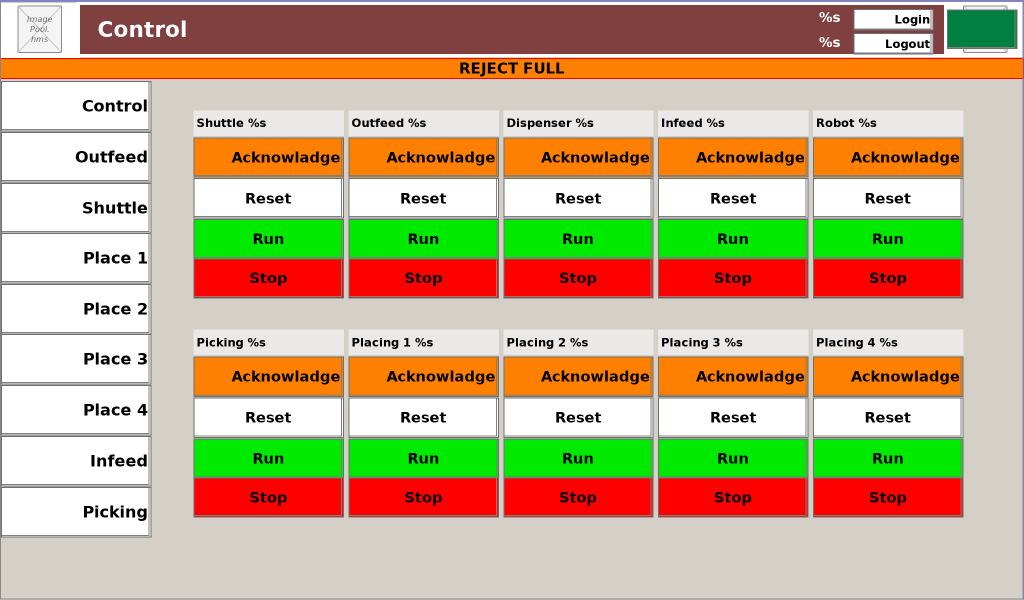
VISUALIZATION Control  // 1024x600
    Frame (0,2 1023x598)
        shows StateMachine()
        shows Test_Outfeed()
        shows Test_Shuttle()
        shows Test_Place1()
        shows Test_Place2()
        shows Test_Place3()
        shows Test_Place4()
        shows Test_Infeed()
        shows Test_Picking()
    Button (1,81 150x50), "Control", image: VisuSymbols.Symbols.Database2
        OnMouseDown: FrameSelectionChange Selection=SelectedFrame=146e207b-fd78-4676-ba16-384fa245d7d2, GlobSel=AssignDir=MainPage.GenElemInst_1003, AssignType=Directly, SelType=Locally
    Button (1,132 150x50), "Outfeed", image: VisuSymbols.Symbols.Database2
        OnMouseDown: FrameSelectionChange Selection=SelectedFrame=146e207b-fd78-4676-ba16-384fa245d7d2, Selection=1, GlobSel=AssignDir=MainPage.GenElemInst_1003, AssignType=Directly, SelType=Locally
    Button (1,183 150x50), "Shuttle", image: VisuSymbols.Symbols.Database2
        OnMouseDown: FrameSelectionChange Selection=SelectedFrame=146e207b-fd78-4676-ba16-384fa245d7d2, Selection=2, GlobSel=AssignDir=MainPage.GenElemInst_1003, AssignType=Directly, SelType=Locally
    Button (1,233 150x50), "Place 1", image: VisuSymbols.Symbols.Database2
        OnMouseDown: FrameSelectionChange Selection=SelectedFrame=146e207b-fd78-4676-ba16-384fa245d7d2, Selection=3, GlobSel=AssignDir=MainPage.GenElemInst_1003, AssignType=Directly, SelType=Locally
    Button (1,284 150x50), "Place 2", image: VisuSymbols.Symbols.Database2
        OnMouseDown: FrameSelectionChange Selection=SelectedFrame=146e207b-fd78-4676-ba16-384fa245d7d2, Selection=4, GlobSel=AssignDir=MainPage.GenElemInst_1003, AssignType=Directly, SelType=Locally
    Button (1,334 150x50), "Place 3", image: VisuSymbols.Symbols.Database2
        OnMouseDown: FrameSelectionChange Selection=SelectedFrame=146e207b-fd78-4676-ba16-384fa245d7d2, Selection=5, GlobSel=AssignDir=MainPage.GenElemInst_1003, AssignType=Directly, SelType=Locally
    Button (1,385 150x50), "Place 4", image: VisuSymbols.Symbols.Database2
        OnMouseDown: FrameSelectionChange Selection=SelectedFrame=146e207b-fd78-4676-ba16-384fa245d7d2, Selection=6, GlobSel=AssignDir=MainPage.GenElemInst_1003, AssignType=Directly, SelType=Locally
    Button (1,436 150x50), "Infeed", image: VisuSymbols.Symbols.Database2
        OnMouseDown: FrameSelectionChange Selection=SelectedFrame=146e207b-fd78-4676-ba16-384fa245d7d2, Selection=7, GlobSel=AssignDir=MainPage.GenElemInst_1003, AssignType=Directly, SelType=Locally
    Button (1,487 150x50), "Picking", image: VisuSymbols.Symbols.Database2
        OnMouseDown: FrameSelectionChange Selection=SelectedFrame=146e207b-fd78-4676-ba16-384fa245d7d2, Selection=8, GlobSel=AssignDir=MainPage.GenElemInst_1003, AssignType=Directly, SelType=Locally
END_VISUALIZATION

// ---- VISUs/TestMode/Test_Infeed.TcVIS
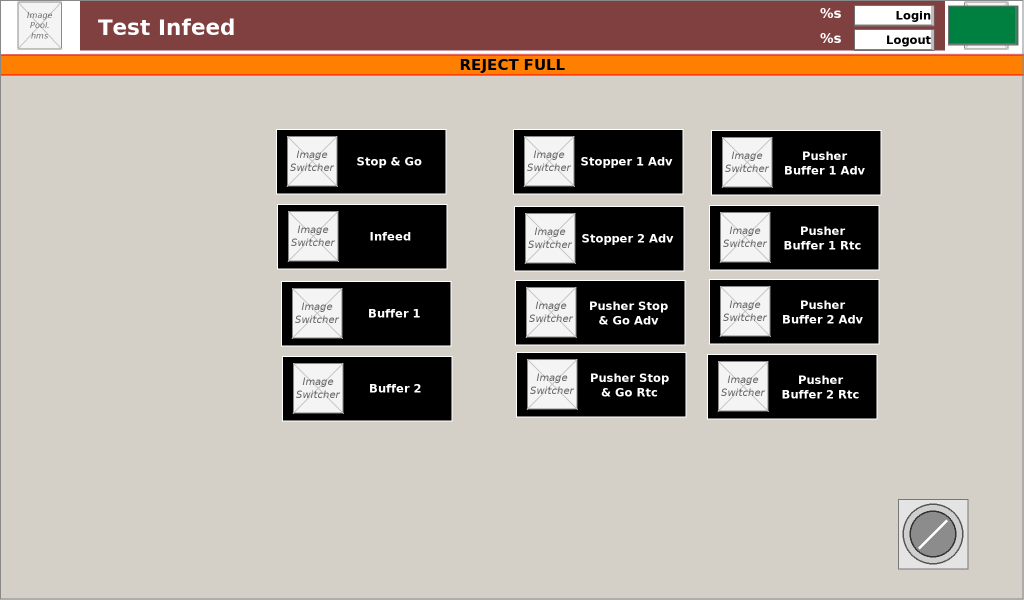
VISUALIZATION Test_Infeed  // 1024x600
    Frame (0,-2 1021x55)
        shows Header()
    Label (95,15 250x25), "Test Infeed"
    RotarySwitch (898,499 70x70), variable: HMI_GVL.bTestModeEnableInfeed, behaviour: TOGGLE, style: Switch-RotarySwitch-Gray
    RoundedRectangle (276,129 170x65)
        toggle HMI_GVL.Test_BoxStopGo_Fwd
    Label (321,149 137x25), "Stop & Go"
    ImageSwitcher (287,136 50x50), variable: HMI_GVL.Test_BoxStopGo_Fwd, behaviour: TOGGLE
    RoundedRectangle (513,129 170x65)
        toggle HMI_GVL.Test_Stopper1
    Label (558,149 137x25), "Stopper 1 Adv"
    ImageSwitcher (524,136 50x50), variable: HMI_GVL.Test_Stopper1, behaviour: TOGGLE
    RoundedRectangle (514,206 170x65)
        toggle HMI_GVL.Test_Stopper2
    Label (559,226 137x25), "Stopper 2 Adv"
    ImageSwitcher (525,213 50x50), variable: HMI_GVL.Test_Stopper2, behaviour: TOGGLE
    RoundedRectangle (277,204 170x65)
        toggle HMI_GVL.Test_BoxInfeed_Fwd
    Label (322,224 137x25), "Infeed"
    ImageSwitcher (288,211 50x50), variable: HMI_GVL.Test_BoxInfeed_Fwd, behaviour: TOGGLE
    RoundedRectangle (281,281 170x65)
        toggle HMI_GVL.Test_BoxBuffer1_Fwd
    Label (326,301 137x25), "Buffer 1"
    ImageSwitcher (292,288 50x50), variable: HMI_GVL.Test_BoxBuffer1_Fwd, behaviour: TOGGLE
    RoundedRectangle (282,356 170x65)
        toggle HMI_GVL.Test_BoxBuffer2_Fwd
    Label (327,376 137x25), "Buffer 2"
    ImageSwitcher (293,363 50x50), variable: HMI_GVL.Test_BoxBuffer2_Fwd, behaviour: TOGGLE
    RoundedRectangle (515,280 170x65)
        toggle HMI_GVL.Test_Pusher_StopGo_Adv
    Label (560,292 137x43), "Pusher Stop & Go Adv"
    ImageSwitcher (526,287 50x50), variable: HMI_GVL.Test_Pusher_StopGo_Adv, behaviour: TOGGLE
    RoundedRectangle (516,352 170x65)
        toggle HMI_GVL.Test_Pusher_StopGo_Rtc
    Label (561,364 137x43), "Pusher Stop & Go Rtc"
    ImageSwitcher (527,359 50x50), variable: HMI_GVL.Test_Pusher_StopGo_Rtc, behaviour: TOGGLE
    RoundedRectangle (711,130 170x65)
        toggle HMI_GVL.Test_Pusher_Buffer1_Adv
    Label (756,142 137x43), "Pusher Buffer 1 Adv"
    ImageSwitcher (722,137 50x50), variable: HMI_GVL.Test_Pusher_Buffer1_Adv, behaviour: TOGGLE
    RoundedRectangle (709,205 170x65)
        toggle HMI_GVL.Test_Pusher_Buffer1_Rtc
    Label (754,217 137x43), "Pusher Buffer 1 Rtc"
    ImageSwitcher (720,212 50x50), variable: HMI_GVL.Test_Pusher_Buffer1_Rtc, behaviour: TOGGLE
    RoundedRectangle (709,279 170x65)
        toggle HMI_GVL.Test_Pusher_Buffer2_Adv
    Label (754,291 137x43), "Pusher Buffer 2 Adv"
    ImageSwitcher (720,286 50x50), variable: HMI_GVL.Test_Pusher_Buffer2_Adv, behaviour: TOGGLE
    RoundedRectangle (707,354 170x65)
        toggle HMI_GVL.Test_Pusher_Buffer2_Rtc
    Label (752,366 137x43), "Pusher Buffer 2 Rtc"
    ImageSwitcher (718,361 50x50), variable: HMI_GVL.Test_Pusher_Buffer2_Rtc, behaviour: TOGGLE
END_VISUALIZATION

// ---- VISUs/TestMode/Test_Place1.TcVIS
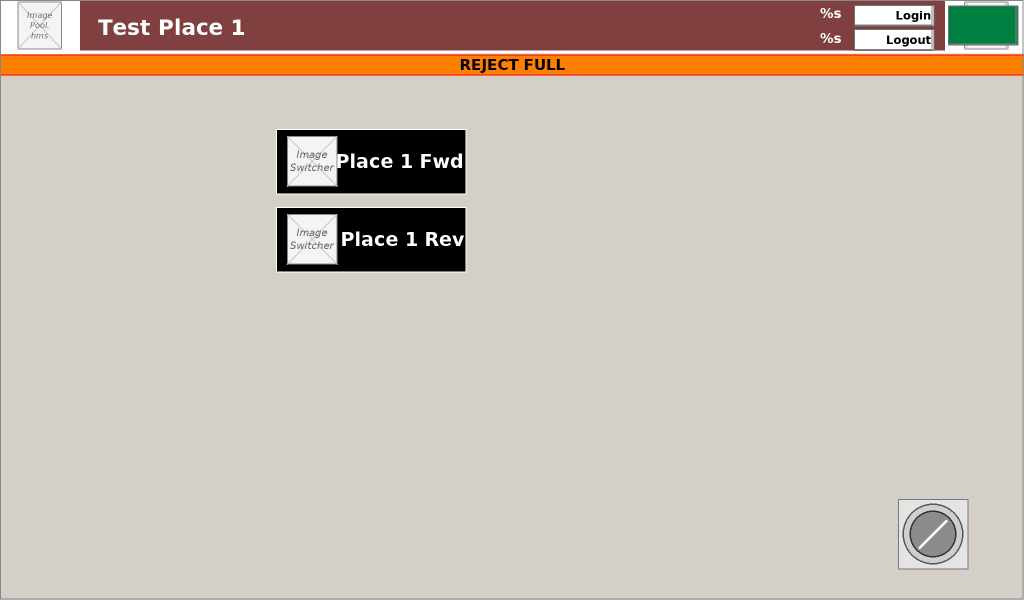
VISUALIZATION Test_Place1  // 1024x600
    Frame (0,-2 1021x55)
        shows Header()
    Label (95,15 250x25), "Test Place 1"
    RotarySwitch (898,499 70x70), variable: HMI_GVL.bTestModeEnablePlacing1, behaviour: TOGGLE, style: Switch-RotarySwitch-Gray
    RoundedRectangle (276,129 190x65)
        toggle Status_GVL.stMotor_Placing1.iTestForward
    Label (331,149 137x25), "Place 1 Fwd"
    ImageSwitcher (287,136 50x50), variable: Status_GVL.stMotor_Placing1.iTestForward, behaviour: TOGGLE
    RoundedRectangle (276,207 190x65)
        toggle Status_GVL.stMotor_Placing1.iTestReverse
    Label (334,227 137x25), "Place 1 Rev"
    ImageSwitcher (287,214 50x50), variable: Status_GVL.stMotor_Placing1.iTestReverse, behaviour: TOGGLE
END_VISUALIZATION

// ---- VISUs/TestMode/Test_Place2.TcVIS
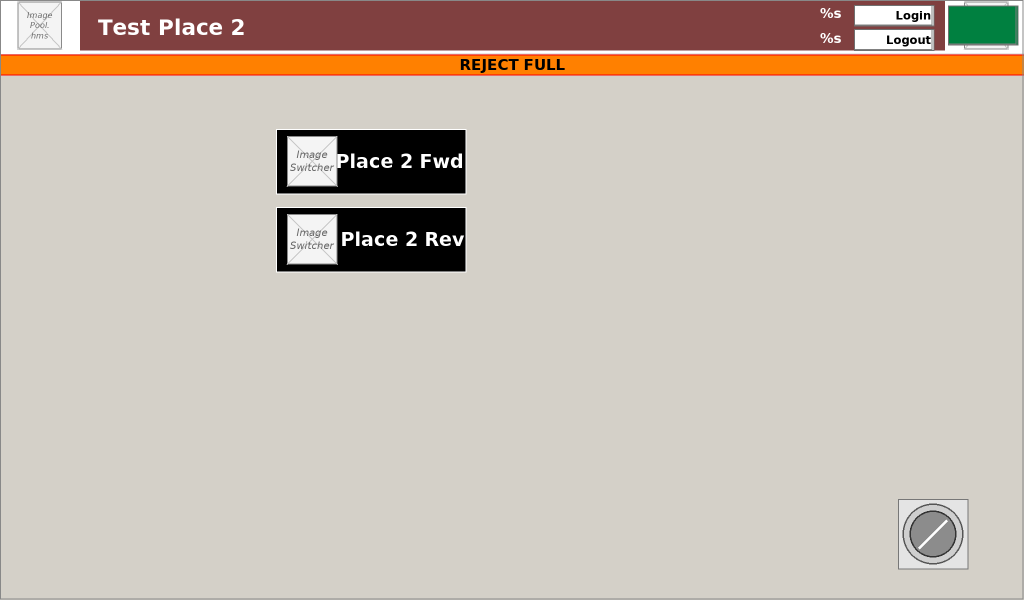
VISUALIZATION Test_Place2  // 1024x600
    Frame (0,-2 1021x55)
        shows Header()
    Label (95,15 250x25), "Test Place 2"
    RotarySwitch (898,499 70x70), variable: HMI_GVL.bTestModeEnablePlacing2, behaviour: TOGGLE, style: Switch-RotarySwitch-Gray
    RoundedRectangle (276,129 190x65)
        toggle Status_GVL.stMotor_Placing2.iTestForward
    Label (331,149 137x25), "Place 2 Fwd"
    ImageSwitcher (287,136 50x50), variable: Status_GVL.stMotor_Placing2.iTestForward, behaviour: TOGGLE
    RoundedRectangle (276,207 190x65)
        toggle Status_GVL.stMotor_Placing2.iTestReverse
    Label (334,227 137x25), "Place 2 Rev"
    ImageSwitcher (287,214 50x50), variable: Status_GVL.stMotor_Placing2.iTestReverse, behaviour: TOGGLE
END_VISUALIZATION

// ---- VISUs/TestMode/Test_Place3.TcVIS
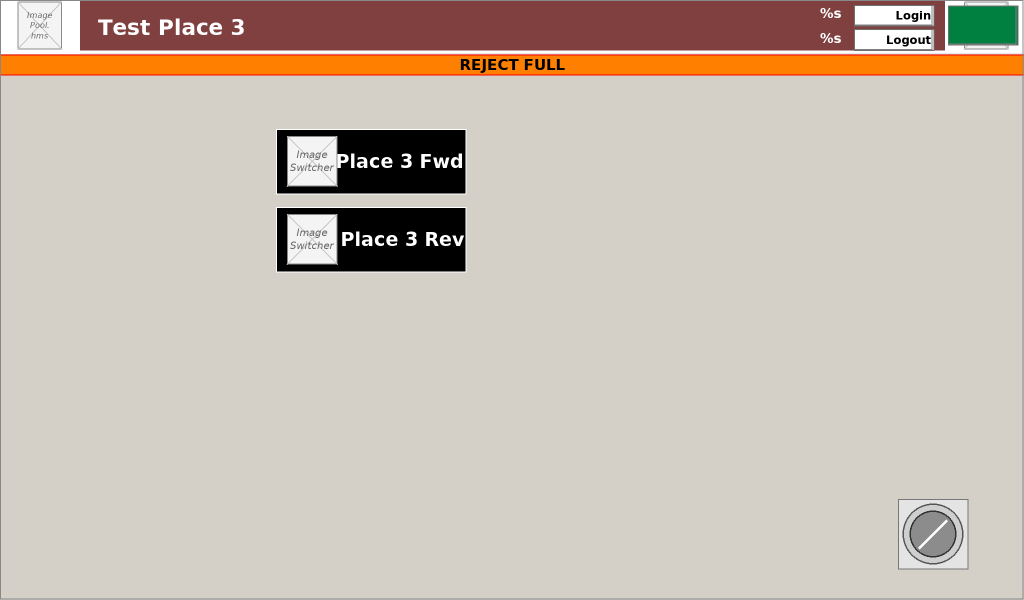
VISUALIZATION Test_Place3  // 1024x600
    Frame (0,-2 1021x55)
        shows Header()
    Label (95,15 250x25), "Test Place 3"
    RotarySwitch (898,499 70x70), variable: HMI_GVL.bTestModeEnablePlacing3, behaviour: TOGGLE, style: Switch-RotarySwitch-Gray
    RoundedRectangle (276,129 190x65)
        toggle Status_GVL.stMotor_Placing3.iTestForward
    Label (331,149 137x25), "Place 3 Fwd"
    ImageSwitcher (287,136 50x50), variable: Status_GVL.stMotor_Placing3.iTestForward, behaviour: TOGGLE
    RoundedRectangle (276,207 190x65)
        toggle Status_GVL.stMotor_Placing3.iTestReverse
    Label (334,227 137x25), "Place 3 Rev"
    ImageSwitcher (287,214 50x50), variable: Status_GVL.stMotor_Placing3.iTestReverse, behaviour: TOGGLE
END_VISUALIZATION

// ---- VISUs/TestMode/Test_Place4.TcVIS
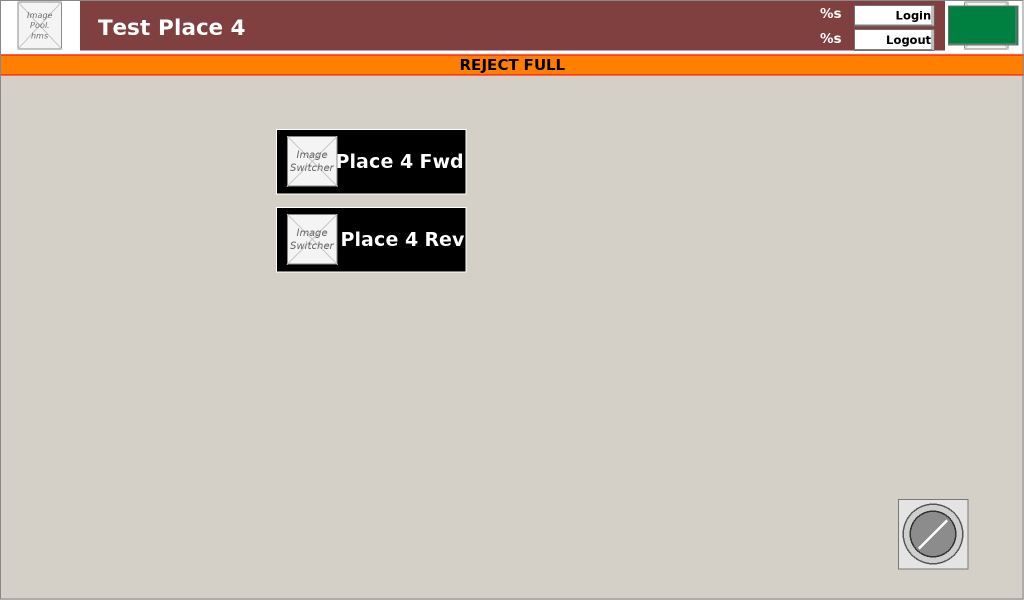
VISUALIZATION Test_Place4  // 1024x600
    Frame (0,-2 1021x55)
        shows Header()
    Label (95,15 250x25), "Test Place 4"
    RotarySwitch (898,499 70x70), variable: HMI_GVL.bTestModeEnablePlacing4, behaviour: TOGGLE, style: Switch-RotarySwitch-Gray
    RoundedRectangle (276,129 190x65)
        toggle Status_GVL.stMotor_Placing4.iTestForward
    Label (331,149 137x25), "Place 4 Fwd"
    ImageSwitcher (287,136 50x50), variable: Status_GVL.stMotor_Placing4.iTestForward, behaviour: TOGGLE
    RoundedRectangle (276,207 190x65)
        toggle Status_GVL.stMotor_Placing4.iTestReverse
    Label (334,227 137x25), "Place 4 Rev"
    ImageSwitcher (287,214 50x50), variable: Status_GVL.stMotor_Placing4.iTestReverse, behaviour: TOGGLE
END_VISUALIZATION

// ---- VISUs/TestMode/Test_Shuttle.TcVIS
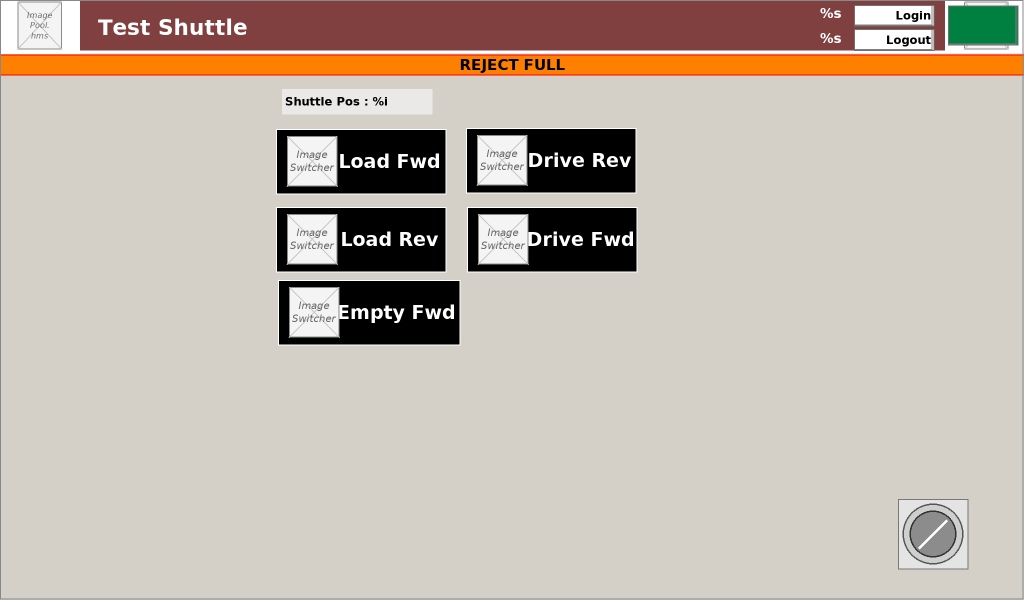
VISUALIZATION Test_Shuttle  // 1024x600
    Frame (0,-2 1021x55)
        shows Header()
    Label (95,15 250x25), "Test Shuttle"
    RotarySwitch (898,499 70x70), variable: HMI_GVL.bTestModeEnableShuttle, behaviour: TOGGLE, style: Switch-RotarySwitch-Gray
    RoundedRectangle (276,129 170x65)
        toggle HMI_GVL.Test_ShuttleLoad_Fwd
    Label (321,149 137x25), "Load Fwd"
    ImageSwitcher (287,136 50x50), variable: HMI_GVL.Test_ShuttleLoad_Fwd, behaviour: TOGGLE
    RoundedRectangle (276,207 170x65)
        toggle HMI_GVL.Test_ShuttleLoad_Rev
    Label (321,227 137x25), "Load Rev"
    ImageSwitcher (287,214 50x50), variable: HMI_GVL.Test_ShuttleLoad_Rev, behaviour: TOGGLE
    RoundedRectangle (278,280 182x65)
        toggle HMI_GVL.Test_ShuttleEmpty_Fwd
    Label (328,300 137x25), "Empty Fwd"
    ImageSwitcher (289,287 50x50), variable: HMI_GVL.Test_ShuttleEmpty_Fwd, behaviour: TOGGLE
    RoundedRectangle (467,207 170x65)
        tap HMI_GVL.Test_ShuttleDrive_Fwd
    Label (512,227 137x25), "Drive Fwd"
    ImageSwitcher (478,214 50x50), variable: HMI_GVL.Test_ShuttleDrive_Fwd, behaviour: TOGGLE
    RoundedRectangle (466,128 170x65)
        tap HMI_GVL.Test_ShuttleDrive_Rev
    Label (511,148 137x25), "Drive Rev"
    ImageSwitcher (477,135 50x50), variable: HMI_GVL.Test_ShuttleDrive_Rev, behaviour: TOGGLE
    Rectangle (282,89 150x25), "Shuttle Pos : %i", text variable: InputOutput_GVL.ShuttlePosition
END_VISUALIZATION

// ---- VISUs/TestMode/Test_Picking.TcVIS
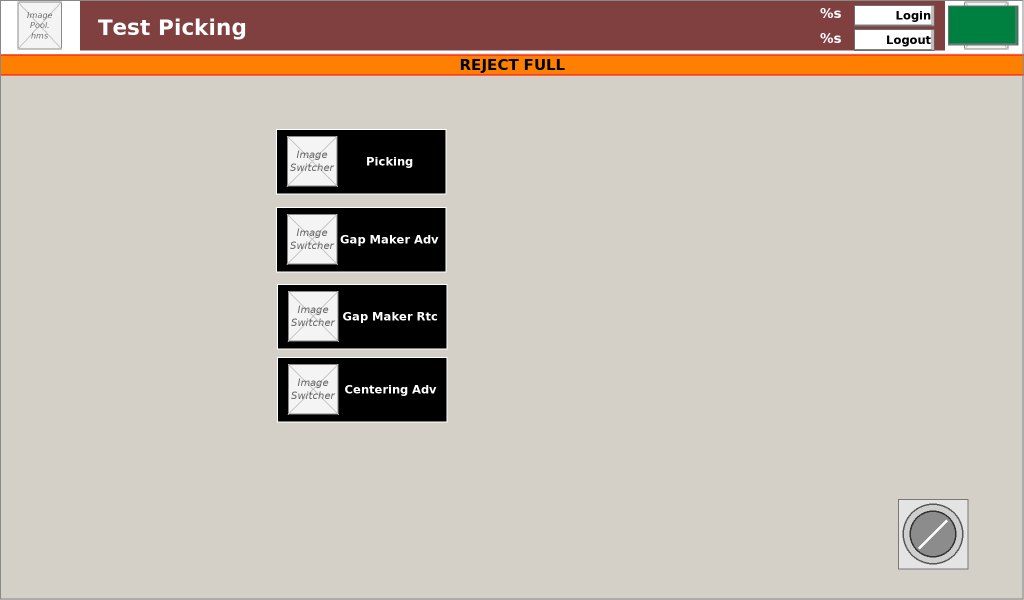
VISUALIZATION Test_Picking  // 1024x600
    Frame (0,-2 1021x55)
        shows Header()
    Label (95,15 250x25), "Test Picking"
    RotarySwitch (898,499 70x70), variable: HMI_GVL.bTestModeEnablePicking, behaviour: TOGGLE, style: Switch-RotarySwitch-Gray
    RoundedRectangle (276,129 170x65)
        toggle Status_GVL.stMotor_Picking.iTestForward
    Label (321,149 137x25), "Picking"
    ImageSwitcher (287,136 50x50), variable: Status_GVL.stMotor_Picking.iTestForward, behaviour: TOGGLE
    RoundedRectangle (276,207 170x65)
        toggle Status_GVL.stPneu_GapMaker.iTestAdvanced
    Label (321,227 137x25), "Gap Maker Adv"
    ImageSwitcher (287,214 50x50), variable: Status_GVL.stPneu_GapMaker.iTestAdvanced, behaviour: TOGGLE
    RoundedRectangle (277,284 170x65)
        toggle Status_GVL.stPneu_GapMaker.iTestRetract
    Label (322,304 137x25), "Gap Maker Rtc"
    ImageSwitcher (288,291 50x50), variable: Status_GVL.stPneu_GapMaker.iTestRetract, behaviour: TOGGLE
    RoundedRectangle (277,357 170x65)
        toggle Status_GVL.stPneu_Centering.iTest
    Label (322,377 137x25), "Centering Adv"
    ImageSwitcher (288,364 50x50), variable: Status_GVL.stPneu_GapMaker.iTestRetract, behaviour: TOGGLE
END_VISUALIZATION
